Staubli VAL3: OnF1.pgx

program OnF1()
  local bool l_bRes
begin
  //
  switch nPage
    case 0
      if sItem!=""
        nPrdIndex=nSelected
        call getList(sProductList[nSelected],sPathList)
        call EditPath()
      else
       popUpMsg("空路径不能编辑")
      endIf

    break
    case 1
      if sItem!=""
        call Path:EditMain(sItem)
      else
        popUpMsg("空路径不能编辑")
      endIf

    break
    //
    case 2
      sNewPath=sItem
      popUpMsg("新增加路径："+sItem)
    break
  endSwitch
  bUserRefresh=bListRefresh=true
end
